// TIA Portal V20 export
DATA_BLOCK "Instance_FB_Read_Data_SR-X100W_Entrace_DB"   // DB106
// stored: AutoNumber false, InstanceOfName FB_Read_Data_SR-X100W, InstanceOfType FB
"FB_Read_Data_SR-X100W"
   // VAR_INPUT
   //    Trigger_Sensor : Bool;
   //    Read_Complete : Bool;
   //    Read_Failure : Bool;
   //    Clear_Data : Bool;
   //    Read_Data_In : "SR-X100W_Read_Data";
   // END_VAR
   // VAR_OUTPUT
   //    Read_Request : Bool;
   //    Read_Complete_Clear : Bool;
   //    Read_Complete_OUT : Bool;
   //    Read_Failure_OUT : Bool;
   //    Read_Data_Out : String[136];
   //    Serial_Number { ExternalAccessible := 'False'; ExternalVisible := 'False'; ExternalWritable := 'False'} : String[17];
   // END_VAR
   // VAR
   //    Aux_Triggger_1 : Bool;
   //    Aux_Triggger_2 : Bool;
   //    Aux_Triggger_3 : Bool;
   //    Aux_Triggger_4 : Bool;
   //    DB_What_Was_Read_Instance { S7_SetPoint := 'True'} : "FB_What_Was_Read";
   //    Timer_Delay_Reset { S7_SetPoint := 'True'} : TON_TIME;
   // END_VAR
BEGIN
END_DATA_BLOCK
